TYPE (* A Structure with 8 BYTES *)
  (* Version 1.0, 2024-02-21, Franz Höpfinger, HR Agrartechnik GmbH *)
  PACKAGE logiBUS::utils::conversion::types;
  ST08B : STRUCT
    B_00 : BYTE; (* BYTE 00 *)
    B_01 : BYTE; (* BYTE 01 *)
    B_02 : BYTE; (* BYTE 02 *)
    B_03 : BYTE; (* BYTE 03 *)
    B_04 : BYTE; (* BYTE 04 *)
    B_05 : BYTE; (* BYTE 05 *)
    B_06 : BYTE; (* BYTE 06 *)
    B_07 : BYTE; (* BYTE 07 *)
  END_STRUCT;
END_TYPE
